TYPE stReciepe :
STRUCT
	_description : STRING(255);
	{attribute addProperty Name "<#Lenght# [mm]>}
	_lenght : stContinuousValueLimits;	
END_STRUCT
END_TYPE

(* stored: Version 1.1.0.1, ProductVersion 3.1.4024.3
   DUT stReciepe: Id {07caa9b1-1592-468b-bd1c-3e869ce6c457} *)
